(* IEC 61131-3 sources: plc_on_fpga_riscv_hybrid/RV_FPGA_PLC_IDE_Projects/xor, 1 file *)

(* ---- xor.il ---- *)
VAR
END_VAR

PROGRAM xor
    d :
        LD     %SW.0
        XOR    %SW.1
        ST     %LEDR.0
END_PROGRAM
